(* IEC 61131-3 sources: eCockpitGit/test_project/src/%F%02 System/%F%03 LoadSaveManager/%POU%FB_LoadSave/%F%Save/%F%Write, 11 files *)

(* ---- %METH%writeBool.st ---- *)
//This adds a value data to the buffer
// |**Version**|**Author**| **Date** |**Changes**
// | 1         | NSN      | 22-06-20 | Creation
METHOD writeBool
VAR_INPUT
	value			:BOOL;				//Address of string for the filler text
END_VAR
(*%!%__DELIMITER__%!%*)
writer.writeBool(value:=value);
logChange(valPoint:=ADR(value),valType:=ESysType.tBool);

(* ---- %METH%writeDint.st ---- *)
//This adds a value data to the buffer
// |**Version**|**Author**| **Date** |**Changes**
// | 1         | NSN      | 22-06-20 | Creation
METHOD writeDint
VAR_INPUT
	value			:DINT;
END_VAR
(*%!%__DELIMITER__%!%*)
writer.writeDint(value:=value);
logChange(valPoint:=ADR(value),valType:=ESysType.tDINT);

(* ---- %METH%writeDword.st ---- *)
//This adds a value data to the buffer
// |**Version**|**Author**| **Date** |**Changes**
// | 1         | NSN      | 16-05-21 | Creation
METHOD writeDword
VAR_INPUT
	value			:DWORD;
END_VAR
(*%!%__DELIMITER__%!%*)
writer.writeDword(value:=value);
logChange(valPoint:=ADR(value),valType:=ESysType.tDWORD);

(* ---- %METH%writeInt.st ---- *)
//This adds a value data to the buffer
// |**Version**|**Author**| **Date** |**Changes**
// | 1         | NSN      | 22-06-20 | Creation
METHOD writeInt
VAR_INPUT
	value			:INT;
END_VAR
(*%!%__DELIMITER__%!%*)
writer.writeInt(value:=value);
logChange(valPoint:=ADR(value),valType:=ESysType.tINT);

(* ---- %METH%writeLint.st ---- *)
//This adds a value data to the buffer
// |**Version**|**Author**| **Date** |**Changes**
// | 1         | NSN      | 22-06-20 | Creation
METHOD writeLint
VAR_INPUT
	value			:LINT;
END_VAR
(*%!%__DELIMITER__%!%*)
writer.writeLint(value:=value);
logChange(valPoint:=ADR(value),valType:=ESysType.tLINT);

(* ---- %METH%writeLword.st ---- *)
//This adds a value data to the buffer
// |**Version**|**Author**| **Date** |**Changes**
// | 1         | NSN      | 16-05-21 | Creation
METHOD writeLword
VAR_INPUT
	value			:LWORD;
END_VAR
(*%!%__DELIMITER__%!%*)
writer.writeLword(value:=value);
logChange(valPoint:=ADR(value),valType:=ESysType.tLWORD);

(* ---- %METH%writeRaw.st ---- *)
//This adds a value data to the buffer
// |**Version**|**Author**| **Date** |**Changes**
// | 1         | NSN      | 22-06-20 | Creation
METHOD writeRaw
VAR_INPUT
	value			:POINTER TO EASCII;	//Address of string for the filler text
END_VAR

(*%!%__DELIMITER__%!%*)
;

(* ---- %METH%writeRawLen.st ---- *)
//Unsupported
METHOD writeRawLen
VAR_INPUT
	value			:POINTER TO EASCII;	//Address of string for the filler text
	len				:DWORD;				//Amount of bytes to write
END_VAR
(*%!%__DELIMITER__%!%*)
;

(* ---- %METH%writeReal.st ---- *)
//This adds a value data to the buffer
// |**Version**|**Author**| **Date** |**Changes**
// | 1         | NSN      | 22-06-20 | Creation
METHOD writeReal
VAR_INPUT
	value			:REAL;
END_VAR
(*%!%__DELIMITER__%!%*)
writer.writeReal(value:=value);
logChange(valPoint:=ADR(value),valType:=ESysType.tREAL);

(* ---- %METH%writeString.st ---- *)
//This adds a value data to the buffer
// |**Version**|**Author**| **Date** |**Changes**
// | 1         | NSN      | 22-06-20 | Creation
METHOD writeString
VAR_INPUT
	value			:POINTER TO EASCII;	//Address of string for the filler text
END_VAR

(*%!%__DELIMITER__%!%*)
writer.writeString(value:=value);
logChange(valPoint:=value,valType:=ESysType.tSTRING);

(* ---- %METH%writeWord.st ---- *)
//This adds a value data to the buffer
// |**Version**|**Author**| **Date** |**Changes**
// | 1         | NSN      | 16-05-21 | Creation
METHOD writeWord
VAR_INPUT
	value			:WORD;
END_VAR
(*%!%__DELIMITER__%!%*)
writer.writeWord(value:=value);
logChange(valPoint:=ADR(value),valType:=ESysType.tWORD);
